# EPICS IOC start-up script: output/git-repo/spk-000cdl_cryo-plc-010/spk_000cdl_cryo_plc_010-test-20220922093722.iocsh
#- @field MODVERSION
#- @runtime YES
#- The version of the PLC-IOC integration

#- @field spk_000cdl_cryo_plc_010_VERSION
#- @runtime YES

#- Load plc interface database
dbLoadRecords("$(DBDIR=)spk_000cdl_cryo_plc_010-test.db", "MODVERSION=$(PLCIOCVERSION)")
